// TIA Portal V17 export
// export: Created 2023-12-22T15:05:25.8877251Z, ExportSetting WithDefaults, DisplayName Totally Integrated Automation Portal, DisplayVersion V17, DisplayName TIA Portal Openness, DisplayVersion V17, DisplayName TIA Portal Version Control Interface, DisplayVersion V17, DisplayName STEP 7 Professional, DisplayVersion V17, DisplayName STEP 7 Safety, DisplayVersion V17, DisplayName WinCC Advanced, DisplayVersion V17
FUNCTION_BLOCK "Block_Pump"   // FB13, LAD
{ S7_Optimized_Access := 'TRUE' }
VERSION : 0.1
// stored: AutoNumber true, IsIECCheckEnabled false, IsRetainMemResEnabled false, MemoryReserve 100, SetENOAutomatically false, UDAEnableTagReadback false
   VAR_INPUT
      All_Lines : Int;
      Status_Pump : Int;
   END_VAR
   VAR_OUTPUT
      Alarm : Bool;
      CMD_Alarm : Bool;
      SP_Result : Real;
   END_VAR
   VAR_IN_OUT
      Start_A : Bool;
   END_VAR
   VAR RETAIN
      PUMP_NUMBER : Int;
      Reserv { S7_SetPoint := 'True'} : Bool;
   END_VAR
   VAR
      Start_Main : Bool;
      Start_Reserv : Bool;
      REQ : Bool;
      REQ_Reserv : Bool;   // Запрос резерва с панели
      pos : Array[0..15] of Bool;
      Events : Word;
   END_VAR
   VAR RETAIN
      Line_Main { S7_SetPoint := 'True'} : Int;
      Line_Reserv { S7_SetPoint := 'True'} : Int;
   END_VAR
   VAR
      T_events : Struct
         SP { ExternalAccessible := 'False'; ExternalVisible := 'False'; ExternalWritable := 'False'} : Int := 3;   // Уставка
         Now { ExternalAccessible := 'False'; ExternalVisible := 'False'; ExternalWritable := 'False'} : Int;   // Текущий счёт
         "Exit" { ExternalAccessible := 'False'; ExternalVisible := 'False'; ExternalWritable := 'False'} : Bool;   // Счёт завершён
         Start { ExternalAccessible := 'False'; ExternalVisible := 'False'; ExternalWritable := 'False'} : Bool;   // Запуск
         Pause { ExternalAccessible := 'False'; ExternalVisible := 'False'; ExternalWritable := 'False'} : Bool;   // Пауза
         Reset { ExternalAccessible := 'False'; ExternalVisible := 'False'; ExternalWritable := 'False'} : Bool;   // Сброс таймера
      END_STRUCT;
   END_VAR
   VAR_TEMP
      ev : Bool;
   END_VAR
   VAR_TEMP   // added for the SCL form of the ladder/FBD networks
      _w1 : Bool;
      _w2 : Bool;
      _w3 : Bool;
      _w4 : Bool;
      _w5 : Bool;
      _w6 : Bool;
      _w7 : Bool;
      _w8 : Bool;
      _w9 : Bool;
      _w10 : Bool;
   END_VAR
BEGIN

REGION Network 1
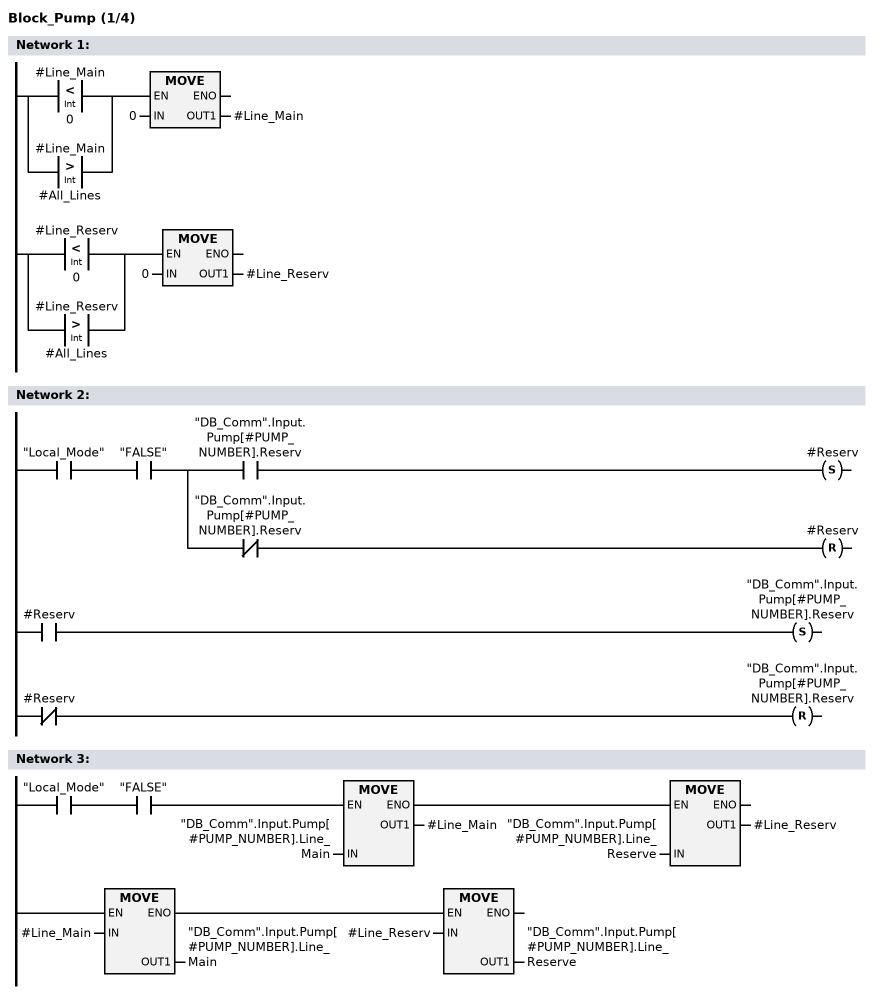
   RUNG wire#powerrail
      { S7_Templates := "SrcType := Int" } LT_Contact(in1 := #Line_Main, in2 := 0)
      wire#w1
      Move(in := 0, out1 => #Line_Main)
   END_RUNG
   RUNG wire#powerrail
      { S7_Templates := "SrcType := Int" } GT_Contact(in1 := #Line_Main, in2 := #All_Lines)
   END_RUNG wire#w1
   RUNG wire#powerrail
      { S7_Templates := "SrcType := Int" } LT_Contact(in1 := #Line_Reserv, in2 := 0)
      wire#w2
      Move(in := 0, out1 => #Line_Reserv)
   END_RUNG
   RUNG wire#powerrail
      { S7_Templates := "SrcType := Int" } GT_Contact(in1 := #Line_Reserv, in2 := #All_Lines)
   END_RUNG wire#w2
   // the same network as SCL:
   IF (#Line_Main < 0) OR (#Line_Main > #All_Lines) THEN #Line_Main := 0; END_IF;
   IF (#Line_Reserv < 0) OR (#Line_Reserv > #All_Lines) THEN #Line_Reserv := 0; END_IF;
END_REGION

REGION Network 2
   RUNG wire#powerrail
      Contact( "Local_Mode" )
      Contact( "FALSE" )
      wire#w1
      Contact( "DB_Comm".Input.Pump[#PUMP_NUMBER].Reserv )
      S_Coil( #Reserv )
   END_RUNG
   RUNG wire#w1
      I_Contact( "DB_Comm".Input.Pump[#PUMP_NUMBER].Reserv )
      R_Coil( #Reserv )
   END_RUNG
   RUNG wire#powerrail
      Contact( #Reserv )
      S_Coil( "DB_Comm".Input.Pump[#PUMP_NUMBER].Reserv )
   END_RUNG
   RUNG wire#powerrail
      I_Contact( #Reserv )
      R_Coil( "DB_Comm".Input.Pump[#PUMP_NUMBER].Reserv )
   END_RUNG
   // the same network as SCL:
   #_w1 := "Local_Mode" AND "FALSE";
   IF #_w1 AND "DB_Comm".Input.Pump[#PUMP_NUMBER].Reserv THEN #Reserv := TRUE; END_IF;
   IF #_w1 AND NOT "DB_Comm".Input.Pump[#PUMP_NUMBER].Reserv THEN #Reserv := FALSE; END_IF;
   IF #Reserv THEN "DB_Comm".Input.Pump[#PUMP_NUMBER].Reserv := TRUE; END_IF;
   IF NOT #Reserv THEN "DB_Comm".Input.Pump[#PUMP_NUMBER].Reserv := FALSE; END_IF;
END_REGION

REGION Network 3
   RUNG wire#powerrail
      Contact( "Local_Mode" )
      Contact( "FALSE" )
      Move(in := "DB_Comm".Input.Pump[#PUMP_NUMBER].Line_Main, out1 => #Line_Main)
      Move(in := "DB_Comm".Input.Pump[#PUMP_NUMBER].Line_Reserve, out1 => #Line_Reserv)
   END_RUNG
   RUNG wire#powerrail
      Move(in := #Line_Main, out1 => "DB_Comm".Input.Pump[#PUMP_NUMBER].Line_Main)
      Move(in := #Line_Reserv, out1 => "DB_Comm".Input.Pump[#PUMP_NUMBER].Line_Reserve)
   END_RUNG
   // the same network as SCL:
   IF "Local_Mode" AND "FALSE" THEN
       #Line_Main := "DB_Comm".Input.Pump[#PUMP_NUMBER].Line_Main;
       #Line_Reserv := "DB_Comm".Input.Pump[#PUMP_NUMBER].Line_Reserve;
   END_IF;
   "DB_Comm".Input.Pump[#PUMP_NUMBER].Line_Main := #Line_Main;
   "DB_Comm".Input.Pump[#PUMP_NUMBER].Line_Reserve := #Line_Reserv;
END_REGION

REGION Network 4: Основной насос
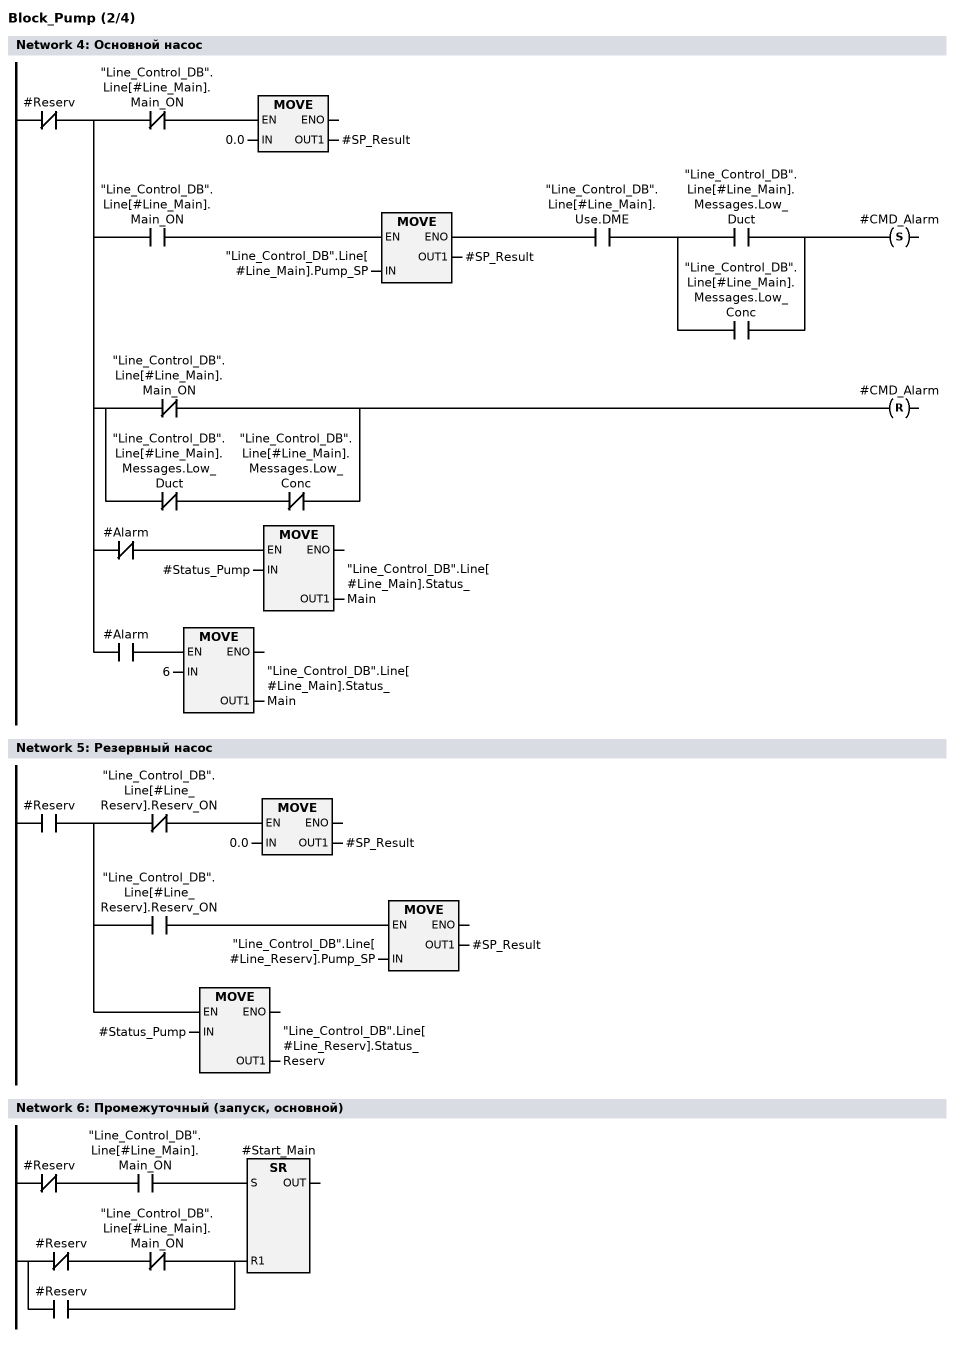
   RUNG wire#powerrail
      I_Contact( #Reserv )
      wire#w1
      I_Contact( "Line_Control_DB".Line[#Line_Main].Main_ON )
      Move(in := 0.0, out1 => #SP_Result)
   END_RUNG
   RUNG wire#w1
      Contact( "Line_Control_DB".Line[#Line_Main].Main_ON )
      Move(in := "Line_Control_DB".Line[#Line_Main].Pump_SP, out1 => #SP_Result)
      Contact( "Line_Control_DB".Line[#Line_Main].Use.DME )
      wire#w2
      Contact( "Line_Control_DB".Line[#Line_Main].Messages.Low_Duct )
      wire#w3
      S_Coil( #CMD_Alarm )
   END_RUNG
   RUNG wire#w2
      Contact( "Line_Control_DB".Line[#Line_Main].Messages.Low_Conc )
   END_RUNG wire#w3
   RUNG wire#w1
      I_Contact( "Line_Control_DB".Line[#Line_Main].Main_ON )
      wire#w4
      R_Coil( #CMD_Alarm )
   END_RUNG
   RUNG wire#w1
      I_Contact( "Line_Control_DB".Line[#Line_Main].Messages.Low_Duct )
      I_Contact( "Line_Control_DB".Line[#Line_Main].Messages.Low_Conc )
   END_RUNG wire#w4
   RUNG wire#w1
      I_Contact( #Alarm )
      Move(in := #Status_Pump, out1 => "Line_Control_DB".Line[#Line_Main].Status_Main)
   END_RUNG
   RUNG wire#w1
      Contact( #Alarm )
      Move(in := 6, out1 => "Line_Control_DB".Line[#Line_Main].Status_Main)
   END_RUNG
   // the same network as SCL:
   IF NOT #Reserv AND NOT "Line_Control_DB".Line[#Line_Main].Main_ON THEN #SP_Result := 0.0; END_IF;
   #_w1 := NOT #Reserv AND "Line_Control_DB".Line[#Line_Main].Main_ON;
   IF #_w1 THEN #SP_Result := "Line_Control_DB".Line[#Line_Main].Pump_SP; END_IF;
   IF #_w1 AND "Line_Control_DB".Line[#Line_Main].Use.DME AND ("Line_Control_DB".Line[#Line_Main].Messages.Low_Duct OR "Line_Control_DB".Line[#Line_Main].Messages.Low_Conc) THEN
       #CMD_Alarm := TRUE;
   END_IF;
   IF NOT #Reserv AND (NOT "Line_Control_DB".Line[#Line_Main].Main_ON OR (NOT "Line_Control_DB".Line[#Line_Main].Messages.Low_Duct AND NOT "Line_Control_DB".Line[#Line_Main].Messages.Low_Conc)) THEN
       #CMD_Alarm := FALSE;
   END_IF;
   IF NOT #Reserv AND NOT #Alarm THEN "Line_Control_DB".Line[#Line_Main].Status_Main := #Status_Pump; END_IF;
   IF NOT #Reserv AND #Alarm THEN "Line_Control_DB".Line[#Line_Main].Status_Main := 6; END_IF;
END_REGION

REGION Network 5: Резервный насос
   RUNG wire#powerrail
      Contact( #Reserv )
      wire#w1
      I_Contact( "Line_Control_DB".Line[#Line_Reserv].Reserv_ON )
      Move(in := 0.0, out1 => #SP_Result)
   END_RUNG
   RUNG wire#w1
      Contact( "Line_Control_DB".Line[#Line_Reserv].Reserv_ON )
      Move(in := "Line_Control_DB".Line[#Line_Reserv].Pump_SP, out1 => #SP_Result)
   END_RUNG
   RUNG wire#w1
      Move(in := #Status_Pump, out1 => "Line_Control_DB".Line[#Line_Reserv].Status_Reserv)
   END_RUNG
   // the same network as SCL:
   IF #Reserv AND NOT "Line_Control_DB".Line[#Line_Reserv].Reserv_ON THEN #SP_Result := 0.0; END_IF;
   IF #Reserv AND "Line_Control_DB".Line[#Line_Reserv].Reserv_ON THEN
       #SP_Result := "Line_Control_DB".Line[#Line_Reserv].Pump_SP;
   END_IF;
   IF #Reserv THEN "Line_Control_DB".Line[#Line_Reserv].Status_Reserv := #Status_Pump; END_IF;
END_REGION

REGION Network 6: Промежуточный (запуск, основной)
   RUNG wire#powerrail
      I_Contact( #Reserv )
      Contact( "Line_Control_DB".Line[#Line_Main].Main_ON )
      S_SR(operand := #Start_Main, r1 := wire#w1)
   END_RUNG
   RUNG wire#powerrail
      I_Contact( #Reserv )
      I_Contact( "Line_Control_DB".Line[#Line_Main].Main_ON )
   END_RUNG wire#w1
   RUNG wire#powerrail
      Contact( #Reserv )
   END_RUNG wire#w1
   // the same network as SCL:
   IF NOT #Reserv AND "Line_Control_DB".Line[#Line_Main].Main_ON THEN
       #Start_Main := TRUE;   // SR flip-flop
   END_IF;
   IF (NOT #Reserv AND NOT "Line_Control_DB".Line[#Line_Main].Main_ON) OR #Reserv THEN
       #Start_Main := FALSE;
   END_IF;
END_REGION

REGION Network 7: Промежуточный (запуск, резервный)
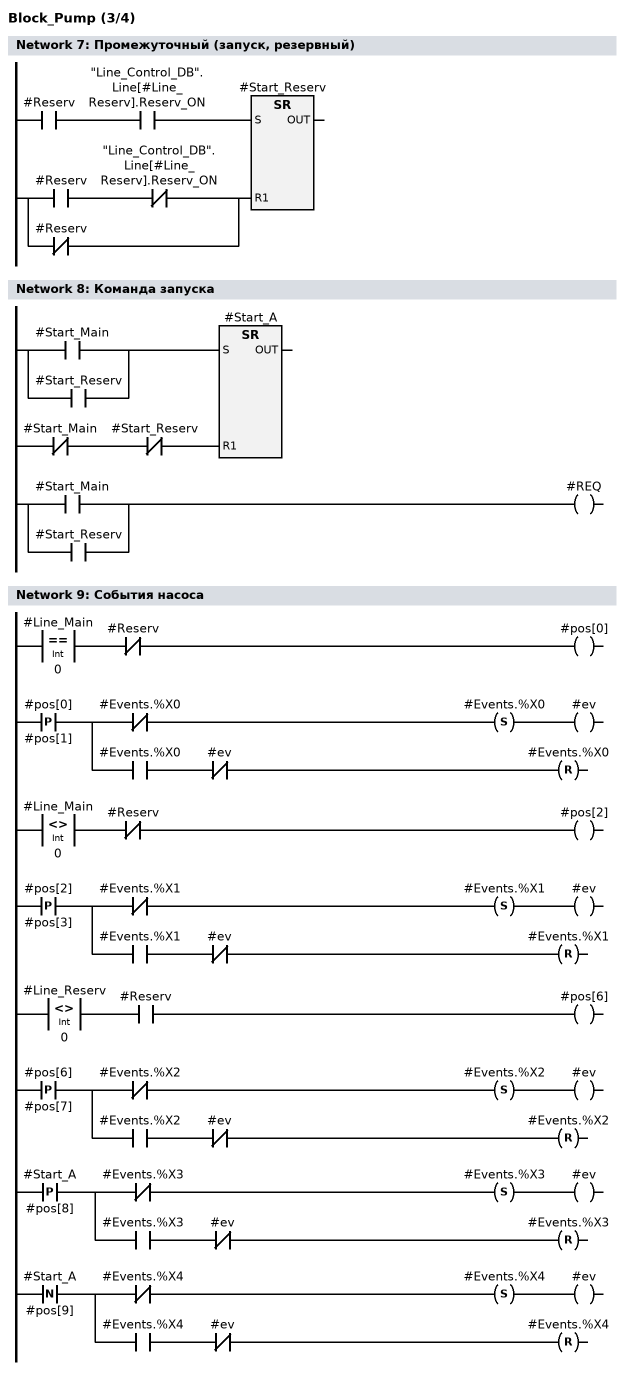
   RUNG wire#powerrail
      Contact( #Reserv )
      Contact( "Line_Control_DB".Line[#Line_Reserv].Reserv_ON )
      S_SR(operand := #Start_Reserv, r1 := wire#w1)
   END_RUNG
   RUNG wire#powerrail
      Contact( #Reserv )
      I_Contact( "Line_Control_DB".Line[#Line_Reserv].Reserv_ON )
   END_RUNG wire#w1
   RUNG wire#powerrail
      I_Contact( #Reserv )
   END_RUNG wire#w1
   // the same network as SCL:
   IF #Reserv AND "Line_Control_DB".Line[#Line_Reserv].Reserv_ON THEN
       #Start_Reserv := TRUE;   // SR flip-flop
   END_IF;
   IF (#Reserv AND NOT "Line_Control_DB".Line[#Line_Reserv].Reserv_ON) OR NOT #Reserv THEN
       #Start_Reserv := FALSE;
   END_IF;
END_REGION

REGION Network 8: Команда запуска
   RUNG wire#powerrail
      Contact( #Start_Main )
      wire#w1
      S_SR(operand := #Start_A, r1 := wire#w2)
   END_RUNG
   RUNG wire#powerrail
      Contact( #Start_Reserv )
   END_RUNG wire#w1
   RUNG wire#powerrail
      I_Contact( #Start_Main )
      I_Contact( #Start_Reserv )
   END_RUNG wire#w2
   RUNG wire#powerrail
      Contact( #Start_Main )
      wire#w3
      Coil( #REQ )
   END_RUNG
   RUNG wire#powerrail
      Contact( #Start_Reserv )
   END_RUNG wire#w3
   // the same network as SCL:
   IF #Start_Main OR #Start_Reserv THEN
       #Start_A := TRUE;   // SR flip-flop
   END_IF;
   IF NOT #Start_Main AND NOT #Start_Reserv THEN #Start_A := FALSE; END_IF;
   #REQ := #Start_Main OR #Start_Reserv;
END_REGION

REGION Network 9: События насоса
   RUNG wire#powerrail
      { S7_Templates := "SrcType := Int" } EQ_Contact(in1 := #Line_Main, in2 := 0)
      I_Contact( #Reserv )
      Coil( #pos[0] )
   END_RUNG
   RUNG wire#powerrail
      P_Contact(operand := #pos[0], bit := #pos[1])
      wire#w1
      I_Contact( #Events.%X0 )
      S_Coil( #Events.%X0 )
      Coil( #ev )
   END_RUNG
   RUNG wire#w1
      Contact( #Events.%X0 )
      I_Contact( #ev )
      R_Coil( #Events.%X0 )
   END_RUNG
   RUNG wire#powerrail
      { S7_Templates := "SrcType := Int" } NE_Contact(in1 := #Line_Main, in2 := 0)
      I_Contact( #Reserv )
      Coil( #pos[2] )
   END_RUNG
   RUNG wire#powerrail
      P_Contact(operand := #pos[2], bit := #pos[3])
      wire#w2
      I_Contact( #Events.%X1 )
      S_Coil( #Events.%X1 )
      Coil( #ev )
   END_RUNG
   RUNG wire#w2
      Contact( #Events.%X1 )
      I_Contact( #ev )
      R_Coil( #Events.%X1 )
   END_RUNG
   RUNG wire#powerrail
      { S7_Templates := "SrcType := Int" } NE_Contact(in1 := #Line_Reserv, in2 := 0)
      Contact( #Reserv )
      Coil( #pos[6] )
   END_RUNG
   RUNG wire#powerrail
      P_Contact(operand := #pos[6], bit := #pos[7])
      wire#w3
      I_Contact( #Events.%X2 )
      S_Coil( #Events.%X2 )
      Coil( #ev )
   END_RUNG
   RUNG wire#w3
      Contact( #Events.%X2 )
      I_Contact( #ev )
      R_Coil( #Events.%X2 )
   END_RUNG
   RUNG wire#powerrail
      P_Contact(operand := #Start_A, bit := #pos[8])
      wire#w4
      I_Contact( #Events.%X3 )
      S_Coil( #Events.%X3 )
      Coil( #ev )
   END_RUNG
   RUNG wire#w4
      Contact( #Events.%X3 )
      I_Contact( #ev )
      R_Coil( #Events.%X3 )
   END_RUNG
   RUNG wire#powerrail
      N_Contact(operand := #Start_A, bit := #pos[9])
      wire#w5
      I_Contact( #Events.%X4 )
      S_Coil( #Events.%X4 )
      Coil( #ev )
   END_RUNG
   RUNG wire#w5
      Contact( #Events.%X4 )
      I_Contact( #ev )
      R_Coil( #Events.%X4 )
   END_RUNG
   // the same network as SCL:
   #pos[0] := (#Line_Main = 0) AND NOT #Reserv;
   #_w1 := #pos[0] AND NOT #pos[1];   // rising edge of #pos[0]
   #pos[1] := #pos[0];
   #_w2 := #_w1 AND NOT #Events.%X0;
   IF #_w2 THEN #Events.%X0 := TRUE; END_IF;
   #ev := #_w2;
   IF #_w1 AND #Events.%X0 AND NOT #ev THEN #Events.%X0 := FALSE; END_IF;
   #pos[2] := (#Line_Main <> 0) AND NOT #Reserv;
   #_w3 := #pos[2] AND NOT #pos[3];   // rising edge of #pos[2]
   #pos[3] := #pos[2];
   #_w4 := #_w3 AND NOT #Events.%X1;
   IF #_w4 THEN #Events.%X1 := TRUE; END_IF;
   #ev := #_w4;
   IF #_w3 AND #Events.%X1 AND NOT #ev THEN #Events.%X1 := FALSE; END_IF;
   #pos[6] := (#Line_Reserv <> 0) AND #Reserv;
   #_w5 := #pos[6] AND NOT #pos[7];   // rising edge of #pos[6]
   #pos[7] := #pos[6];
   #_w6 := #_w5 AND NOT #Events.%X2;
   IF #_w6 THEN #Events.%X2 := TRUE; END_IF;
   #ev := #_w6;
   IF #_w5 AND #Events.%X2 AND NOT #ev THEN #Events.%X2 := FALSE; END_IF;
   #_w7 := #Start_A AND NOT #pos[8];   // rising edge of #Start_A
   #pos[8] := #Start_A;
   #_w8 := #_w7 AND NOT #Events.%X3;
   IF #_w8 THEN #Events.%X3 := TRUE; END_IF;
   #ev := #_w8;
   IF #_w7 AND #Events.%X3 AND NOT #ev THEN #Events.%X3 := FALSE; END_IF;
   #_w9 := NOT #Start_A AND #pos[9];   // falling edge of #Start_A
   #pos[9] := #Start_A;
   #_w10 := #_w9 AND NOT #Events.%X4;
   IF #_w10 THEN #Events.%X4 := TRUE; END_IF;
   #ev := #_w10;
   IF #_w9 AND #Events.%X4 AND NOT #ev THEN #Events.%X4 := FALSE; END_IF;
END_REGION

REGION Network 10
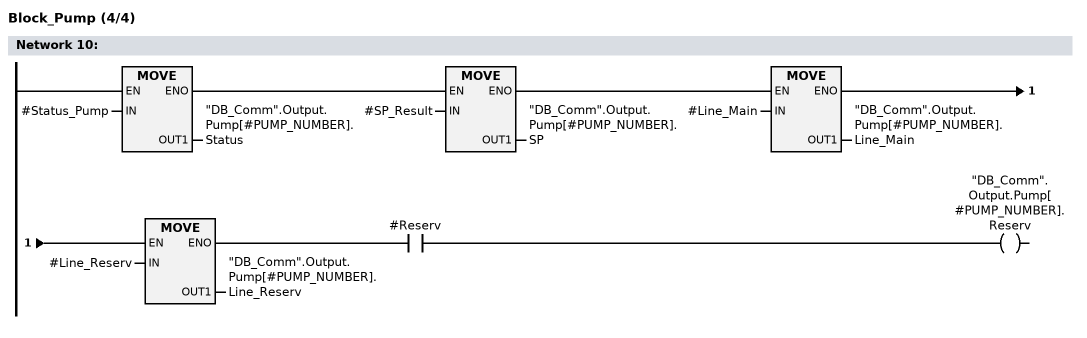
   RUNG wire#powerrail
      Move(in := #Status_Pump, out1 => "DB_Comm".Output.Pump[#PUMP_NUMBER].Status)
      Move(in := #SP_Result, out1 => "DB_Comm".Output.Pump[#PUMP_NUMBER].SP)
      Move(in := #Line_Main, out1 => "DB_Comm".Output.Pump[#PUMP_NUMBER].Line_Main)
      Move(in := #Line_Reserv, out1 => "DB_Comm".Output.Pump[#PUMP_NUMBER].Line_Reserv)
      Contact( #Reserv )
      Coil( "DB_Comm".Output.Pump[#PUMP_NUMBER].Reserv )
   END_RUNG
   // the same network as SCL:
   "DB_Comm".Output.Pump[#PUMP_NUMBER].Status := #Status_Pump;
   "DB_Comm".Output.Pump[#PUMP_NUMBER].SP := #SP_Result;
   "DB_Comm".Output.Pump[#PUMP_NUMBER].Line_Main := #Line_Main;
   "DB_Comm".Output.Pump[#PUMP_NUMBER].Line_Reserv := #Line_Reserv;
   "DB_Comm".Output.Pump[#PUMP_NUMBER].Reserv := #Reserv;
END_REGION
END_FUNCTION_BLOCK
